PROGRAM Sequence  //make sure the change the name to Sequence when we use it for the HMI bitmappings.
VAR
	AverageTemp		: REAL := 0;
	Sum				: REAL := 0;;
	i				: INT := 1;
	n				: INT := 12;
	NumOfTherm		: UINT := 12;
END_VAR


//find sum
FOR i := 1 TO n BY 1 DO 
	
	Sum := Sum + MCP_IO.ThermalCouple[i].TemperatureFB;

END_FOR
	
NumOfTherm.0 := HMI_DB.ThermalCouple[1].IncludeSW;
NumOfTherm.1 := HMI_DB.ThermalCouple[2].IncludeSW;
NumOfTherm.2 := HMI_DB.ThermalCouple[3].IncludeSW;
NumOfTherm.3 := HMI_DB.ThermalCouple[4].IncludeSW;
NumOfTherm.4 := HMI_DB.ThermalCouple[5].IncludeSW;
NumOfTherm.5 := HMI_DB.ThermalCouple[6].IncludeSW;
NumOfTherm.6 := HMI_DB.ThermalCouple[7].IncludeSW;
NumOfTherm.7 := HMI_DB.ThermalCouple[8].IncludeSW;
NumOfTherm.8 := HMI_DB.ThermalCouple[9].IncludeSW;
NumOfTherm.9 := HMI_DB.ThermalCouple[10].IncludeSW;
NumOfTherm.10 := HMI_DB.ThermalCouple[11].IncludeSW;
NumOfTherm.11 := HMI_DB.ThermalCouple[12].IncludeSW;


//USED AS FEEDBACK
AverageTemp := Sum/NumOfTherm;



//PRG_FB_CTRL_PID();


IF i > n THEN
	i := 1;
END_IF

END_PROGRAM

(* stored: Version 1.1.0.1, ProductVersion 3.1.4024.11
   POU Sequence: Id {b02178e8-8fb0-42cf-905a-18f03fa2724e}, SpecialFunc None *)
